// TIA Portal V17 export
// export: Created 2022-03-12T16:05:31.8431672Z, ExportSetting WithDefaults, DisplayName Totally Integrated Automation Portal, DisplayVersion V17, DisplayName TIA Portal Openness, DisplayVersion V17, DisplayName TIA Portal Version Control Interface, DisplayVersion V17, DisplayName STEP 7 Professional, DisplayVersion V17, DisplayName STEP 7 Safety, DisplayVersion V17, DisplayName WinCC Advanced / Unified PC, DisplayVersion V17
DATA_BLOCK "RecipeManagement"   // DB31618
TITLE = CPG_RecipeManagement
{ S7_Optimized_Access := 'TRUE' }
AUTHOR : tech.team.motioncontrol@siemens.com
FAMILY : CPG
VERSION : 1.1
// Support: tech.team.motioncontrol@siemens.com
// stored: AutoNumber true, DBAccessibleFromOPCUA true, DBAccessibleFromWebserver true, IsOnlyStoredInLoadMemory false, IsRetainMemResEnabled false, IsWriteProtectedInAS false, MemoryReserve 0
   VAR
      HMI_Command : Struct   // Helper bits for HMI Recipe Control
         Change : Struct
            changeCmd : Bool;
            changeID : Int;
            cancel : Bool;
            request : Bool;
         END_STRUCT;
         Save : Struct
            saveCmd : Bool;
            saveAsCmd : Bool;
            saveAsDestinationID : Int;
            saveAsNewName : String[60];
            cancel : Bool;
            request : Bool;
         END_STRUCT;
         Copy : Struct
            copyCmd : Bool;
            copySourceID : Int;
            copyDestinationID : Int;
            copyNewName : String[60];
            cancel : Bool;
            request : Bool;
         END_STRUCT;
         Delete : Struct
            deleteCmd : Bool;
            deleteID : Int;
            cancel : Bool;
            request : Bool;
         END_STRUCT;
         resetAllTimes : Bool;
      END_STRUCT;
      HMI_Indicator : Struct   // Helper bits for HMI Recipe Control
         changeConfirm : Bool;
         saveAsConfirm : Bool;
         copyConfirm : Bool;
         deleteConfirm : Bool;
         changeErr : Bool;
         saveAsErr : Bool;
         copyErr : Bool;
         deleteErr : Bool;
      END_STRUCT;
      setpointsArray_REAL { S7_SetPoint := 'True'} : Array[0..11] of "CPG_typeRecipeSetpoint_REAL";   // The setpoints that are displayed
      setpointsArray_DINT { S7_SetPoint := 'True'} : Array[0..11] of "CPG_typeRecipeSetpoint_DINT";   // The setpoints that are displayed
      setpointsArray_BOOL { S7_SetPoint := 'True'} : Array[0..11] of "CPG_typeRecipeSetpoint_BOOL";   // The setpoints that are displayed
      setpointsArray_STRING { S7_SetPoint := 'True'} : Array[0..11] of "CPG_typeRecipeSetpoint_STRING";   // The setpoints that are displayed
      setpointPopup_REAL { S7_SetPoint := 'True'} : "CPG_typeRecipeSetpoint_REAL";   // The setpoint in the popup
      setpointPopup_DINT { S7_SetPoint := 'True'} : "CPG_typeRecipeSetpoint_DINT";   // The setpoint in the popup
      setpointPopup_BOOL { S7_SetPoint := 'True'} : "CPG_typeRecipeSetpoint_BOOL";   // The setpoint in the popup
      setpointPopup_STRING { S7_SetPoint := 'True'} : "CPG_typeRecipeSetpoint_STRING";   // The setpoint in the popup
      popupTrackers : Array[0..3] of Int;   // Int to track the location of popup
      currentPages : Array[0..4] of Int;   // Current page of setpoints (or recipes)
      maxPages : Array[0..4] of Int;   // Max page of setpoints (or recipes)
      displayDisable_REAL : Array[0..11] of Bool;   // True if that setpoint should be hidden
      displayDisable_DINT : Array[0..11] of Bool;   // True if that setpoint should be hidden
      displayDisable_BOOL : Array[0..11] of Bool;   // True if that setpoint should be hidden
      displayDisable_STRING : Array[0..11] of Bool;   // True if that setpoint should be hidden
      recipeArrayNames : Array[0..19] of String[60];   // Recipe names to display
      recipeArraySaves : Array[0..19] of DTL;   // Recipe times to display
      recipeArrayTimes : Array[0..19] of Time;   // Recipe savepoints to display
      recipeArrayNums : Array[0..19] of Int;   // Recipe numbers
      recipeArrayHide : Array[0..19] of Bool;   // True if that recipe should be hidden
   END_VAR
BEGIN
   currentPages[0..4] := 1;
   maxPages[0..3] := 1;
END_DATA_BLOCK
